FUNCTION_BLOCK SUBL_0 (* Event-only Local Group Subscriber *)
  (* Standard: 61499-1; Classification: Communications; Description: Local Event Group Subscriber *)
  (* Version 0.1, 2002-05-02, JHC, Rockwell Automation, Optimized. *)
  (* Version 0.0, 2001-10-02, JHC, Rockwell Automation, Copied/modified from SUBSCRIBE *)
  (* Compiler header: package fb.rt.net; *)
  (* Compiler Java IBM VisualAge 3.0 *)
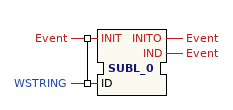
  EVENT_INPUT
    INIT WITH ID; (* Service Initialization *)
  END_EVENT
  EVENT_OUTPUT
    INITO; (* Initialization Confirm *)
    IND; (* Service Indication *)
  END_EVENT
  VAR_INPUT
    ID : WSTRING; (* Local Group Name-Default is FB Instance Name *)
  END_VAR
END_FUNCTION_BLOCK
